// TIA Portal V19 export
DATA_BLOCK "MANUAL BIT"   // DB4
{ S7_Optimized_Access := 'FALSE' }
   VAR
      "P-202 A RO 1 FEED PUMP" : Bool;
      "P-202 B RO 1 FEED PUMP" : Bool;
      "P-202 C RO 1 FEED PUMP" : Bool;
      "P-301 A RO 1 HPP PUMP" : Bool;
      "P-301 B RO 1 HPP PUMP" : Bool;
      "P-401 A RO 2 FEED PUMP" : Bool;
      "P-401 B RO 2 FEED PUMP" : Bool;
      "P-401 C RO 2 FEED PUMP" : Bool;
      "P-402  A RO 2 HPP" : Bool;
      "P-402 B" : Bool;
      "P-501 A EDI FEED PUMP" : Bool;
      "P-501 B EDI FEED PUMP" : Bool;
      "P-501 C EDI FEED PUMP" : Bool;
      "EDI 501" : Bool;
      "EDI 502" : Bool;
      "DP 703" : Bool;
      "DP 704" : Bool;
      "DP 705" : Bool;
      "ABV 301" : Bool;
      "ABV 302" : Bool;
      "AGLV-301" : Bool;
      "AGLV-302" : Bool;
      "AGLV-401" : Bool;
      "AGLV-402" : Bool;
      "AGLV-501" : Bool;
      "AGLV-502" : Bool;
      "SPARE 13" : Bool;
      "SPARE 16" : Bool;
      "SPARE 17" : Bool;
      "SPARE 18" : Bool;
      "SPARE 19" : Bool;
      "SPARE 20" : Bool;
      "SPARE 21" : Bool;
      "SPARE 22" : Bool;
      "SPARE 23" : Bool;
      "SPARE 24" : Bool;
      "SPARE 25" : Bool;
      "SPARE 26" : Bool;
      "SPARE 27" : Bool;
      "SPARE 28" : Bool;
      "SPARE 29" : Bool;
      "SPARE 30" : Bool;
   END_VAR
BEGIN
END_DATA_BLOCK
